FUNCTION_BLOCK FB_Part207ParametersLED
VAR_INPUT
	ipDALICommunication											:	I_DALICommunication;
END_VAR
VAR_OUTPUT
	bBusy														:	BOOL;
END_VAR
VAR
	{region "Visu"}
	bRead														:	BOOL;
	{endregion}
	nStep														:	INT;
	nAddress													:	BYTE;
	nFeatures													:	BYTE;
	bQueryShortCircuitEnabled									:	BOOL;
	bQueryIdleTimeDetectionEnabled								:	BOOL;
	bQueryLoadDecreaseEnabled									:	BOOL;
	bQueryLoadIncreaseEnabled									:	BOOL;
	bQueryCurrentProtectionDevicePresent						:	BOOL;
	bQueryThermalSwitchEnabled									:	BOOL;
	bQueryReductionOfLuminouFluxRegardingThermalOverloadEnabled	:	BOOL;
	bPhysicalSelectionSupported             					:	BOOL;
	bLEDPowerSupply              								:	BOOL;
	bLEDModule													:	BOOL;
	bACSupply               									:	BOOL;
	bDCSupply               									:	BOOL;
	bPWMOperation              									:	BOOL;
	bAMOperation               									:	BOOL;
	bOutputCurrentControlled									:	BOOL;
	bPowerPulseOperation										:	BOOL;

	bHideWaitSymbol												:	BOOL := TRUE;
	bInvisible													:	BOOL := TRUE; // Variable to hide Parameters which are currently not covered by certified device types.

	fb207QueryFeatures 											:	FB_DALI207QueryFeatures(0);
END_VAR

{region "Detect Commands"}
IF (bRead AND (nStep = 0)) THEN
	nStep := 10;
	bRead := FALSE;
	bHideWaitSymbol := FALSE;
END_IF

{endregion}
{region "Manage Dialog Selection}
IF (nStep = 0) THEN
	bBusy := FALSE;
ELSE
	bBusy := TRUE;
END_IF
{endregion}
{region "Execute Commands"}
CASE nStep OF
0:
{region "Init"}
	bRead := FALSE;
	bHideWaitSymbol := TRUE;

	fb207QueryFeatures.ipDALICommunication := ipDALICommunication;
{endregion}
{region "Read"}
10:
{region "Query Features"}
	fb207QueryFeatures(bStart := TRUE,
					   nAddress := nAddress,
					   eAddressType := Tc3_DALI.E_DALIAddressType.Short,
					   eCommandPriority := Tc3_DALI.E_DALICommandPriority.Middle,
					   nFeatures=> nFeatures);

	IF (NOT fb207QueryFeatures.bBusy) THEN
		fb207QueryFeatures(bStart := FALSE);
		bQueryShortCircuitEnabled := nFeatures.0;
		bQueryIdleTimeDetectionEnabled := nFeatures.1;
		bQueryLoadDecreaseEnabled := nFeatures.2;
		bQueryLoadIncreaseEnabled := nFeatures.3;
		bQueryCurrentProtectionDevicePresent := nFeatures.4;
		bQueryThermalSwitchEnabled := nFeatures.5;
		bQueryReductionOfLuminouFluxRegardingThermalOverloadEnabled := nFeatures.6;
		bPhysicalSelectionSupported := nFeatures.7;
		nStep := 0;
	END_IF
{endregion}
{endregion}
END_CASE

END_FUNCTION_BLOCK

(* stored: Version 1.1.0.1, ProductVersion 3.1.4024.10
   POU FB_Part207ParametersLED: Id {7f76f42e-2064-4c62-8d2f-d827dadf3e86}, SpecialFunc None *)
